PROGRAM MAIN
VAR
END_VAR

DALI_Commissioning();

END_PROGRAM

(* stored: Version 1.1.0.1, ProductVersion 3.1.4024.10
   POU MAIN: Id {a47f7a2e-fd82-49d8-b01d-2a458ed98686}, SpecialFunc None *)
